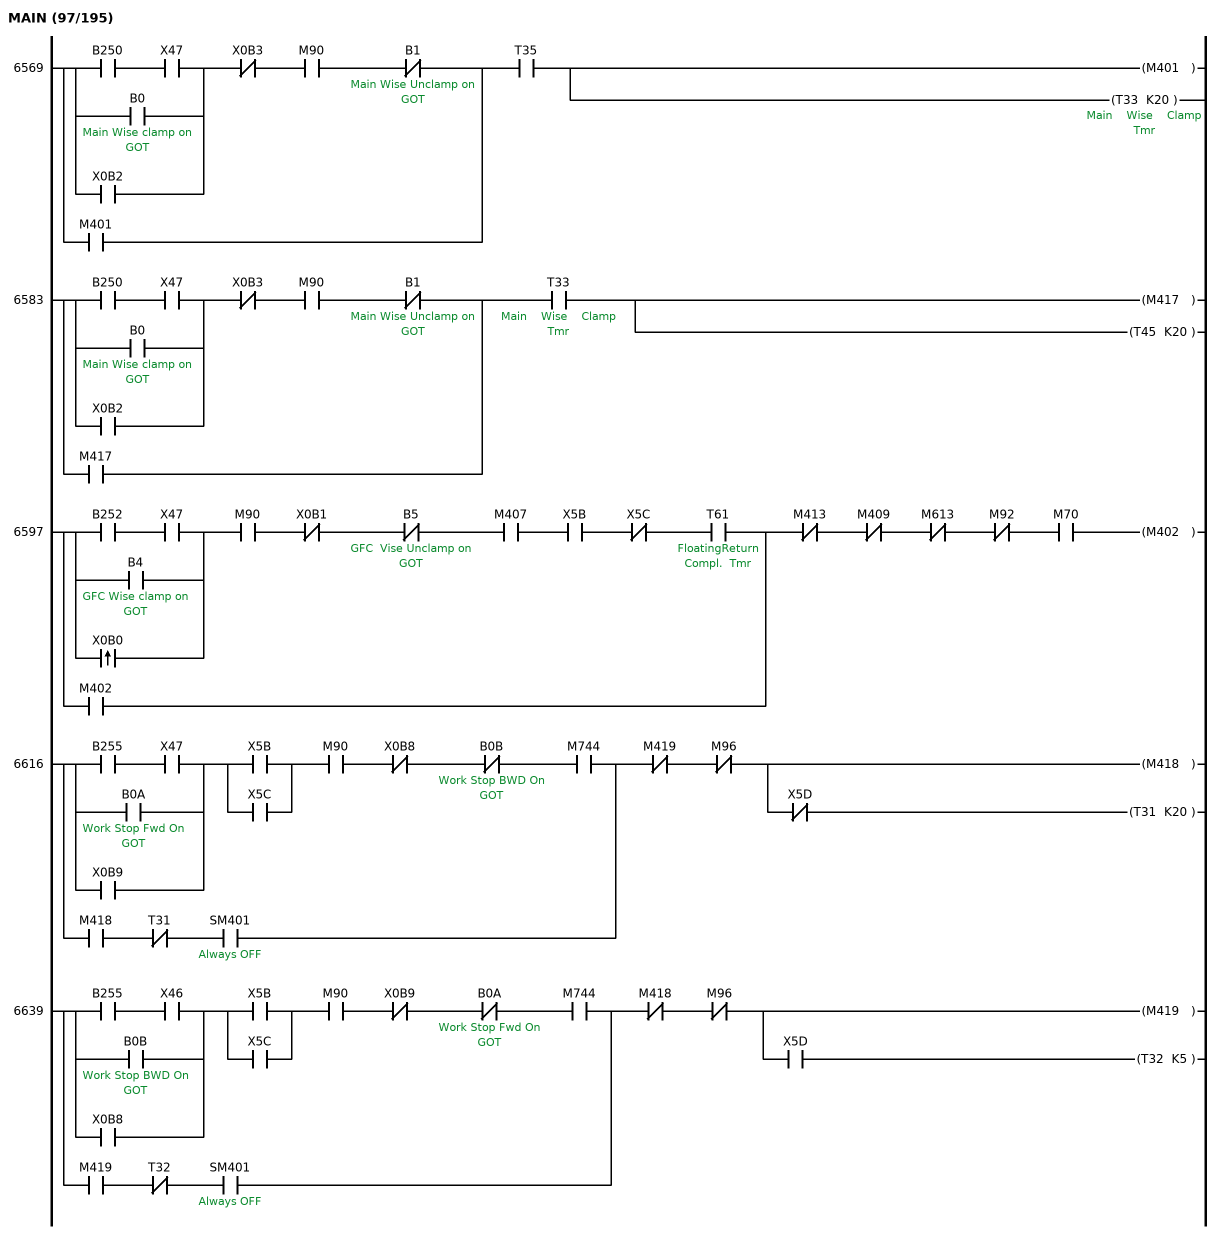
[picture p96: ladder of MAIN, rungs at steps 6569 to 6639]
6569  LD      B250
      AND     X47
      OR      B0  ; Main Wise clamp on GOT
      OR      X0B2
      ANI     X0B3
      AND     M90
      ANI     B1  ; Main Wise Unclamp on GOT
      OR      M401
      AND     T35
      OUT     M401
      OUT     T33 K20  ; Main    Wise    Clamp   Tmr
6583  LD      B250
      AND     X47
      OR      B0  ; Main Wise clamp on GOT
      OR      X0B2
      ANI     X0B3
      AND     M90
      ANI     B1  ; Main Wise Unclamp on GOT
      OR      M417
      AND     T33  ; Main    Wise    Clamp   Tmr
      OUT     M417
      OUT     T45 K20
6597  LD      B252
      AND     X47
      OR      B4  ; GFC Wise clamp on GOT
      ORP     X0B0
      AND     M90
      ANI     X0B1
      ANI     B5  ; GFC  Vise Unclamp on GOT
      AND     M407
      AND     X5B
      ANI     X5C
      AND     T61  ; FloatingReturn  Compl.  Tmr
      OR      M402
      ANI     M413
      ANI     M409
      ANI     M613
      ANI     M92
      AND     M70
      OUT     M402
6616  LD      B255
      AND     X47
      OR      B0A  ; Work Stop Fwd On GOT
      OR      X0B9
      LD      X5B
      OR      X5C
      ANB
      AND     M90
      ANI     X0B8
      ANI     B0B  ; Work Stop BWD On GOT
      AND     M744
      LD      M418
      ANI     T31
      AND     SM401  ; Always OFF
      ORB
      ANI     M419
      ANI     M96
      OUT     M418
      ANI     X5D
      OUT     T31 K20
6639  LD      B255
      AND     X46
      OR      B0B  ; Work Stop BWD On GOT
      OR      X0B8
      LD      X5B
      OR      X5C
      ANB
      AND     M90
      ANI     X0B9
      ANI     B0A  ; Work Stop Fwd On GOT
      AND     M744
      LD      M419
      ANI     T32
      AND     SM401  ; Always OFF
      ORB
      ANI     M418
      ANI     M96
      OUT     M419
      AND     X5D
      OUT     T32 K5
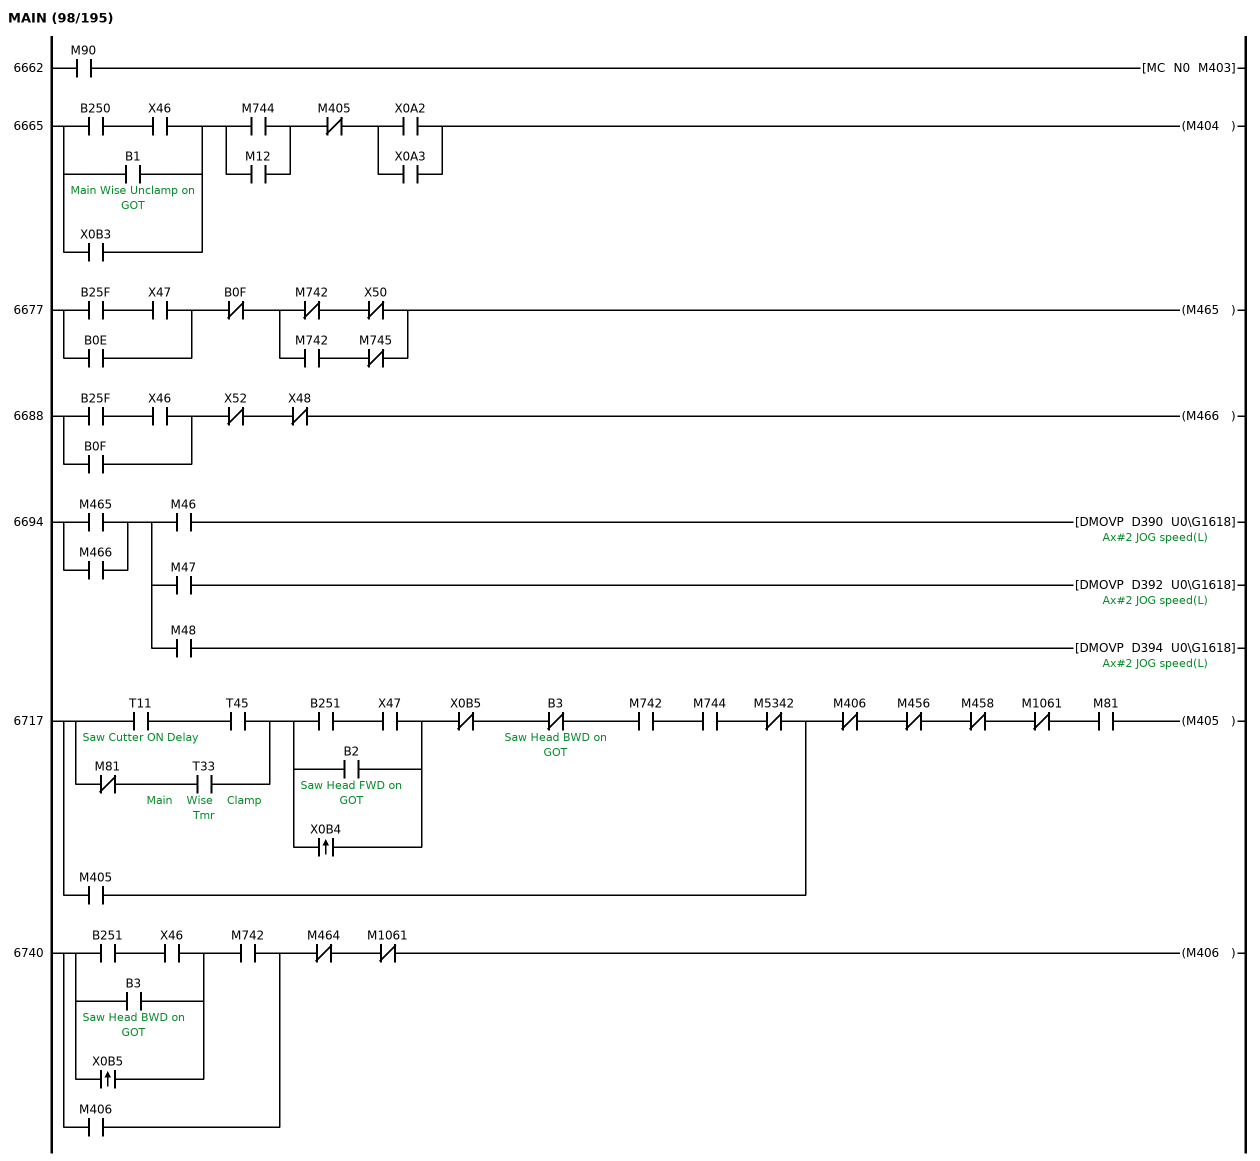
6662  LD      M90
      MC      N0 M403
6665  LD      B250
      AND     X46
      OR      B1  ; Main Wise Unclamp on GOT
      OR      X0B3
      LD      M744
      OR      M12
      ANB
      ANI     M405
      LD      X0A2
      OR      X0A3
      ANB
      OUT     M404
6677  LD      B25F
      AND     X47
      OR      B0E
      ANI     B0F
      LDI     M742
      ANI     X50
      LD      M742
      ANI     M745
      ORB
      ANB
      OUT     M465
6688  LD      B25F
      AND     X46
      OR      B0F
      ANI     X52
      ANI     X48
      OUT     M466
6694  LD      M465
      OR      M466
      MPS
      AND     M46
      DMOVP   D390 U0\G1618
      MRD
      AND     M47
      DMOVP   D392 U0\G1618
      MPP
      AND     M48
      DMOVP   D394 U0\G1618
6717  LD      T11  ; Saw Cutter ON Delay
      AND     T45
      LDI     M81
      AND     T33  ; Main    Wise    Clamp   Tmr
      ORB
      LD      B251
      AND     X47
      OR      B2  ; Saw Head FWD on GOT
      ORP     X0B4
      ANB
      ANI     X0B5
      ANI     B3  ; Saw Head BWD on GOT
      AND     M742
      AND     M744
      ANI     M5342
      OR      M405
      ANI     M406
      ANI     M456
      ANI     M458
      ANI     M1061
      AND     M81
      OUT     M405
6740  LD      B251
      AND     X46
      OR      B3  ; Saw Head BWD on GOT
      ORP     X0B5
      AND     M742
      OR      M406
      ANI     M464
      ANI     M1061
      OUT     M406
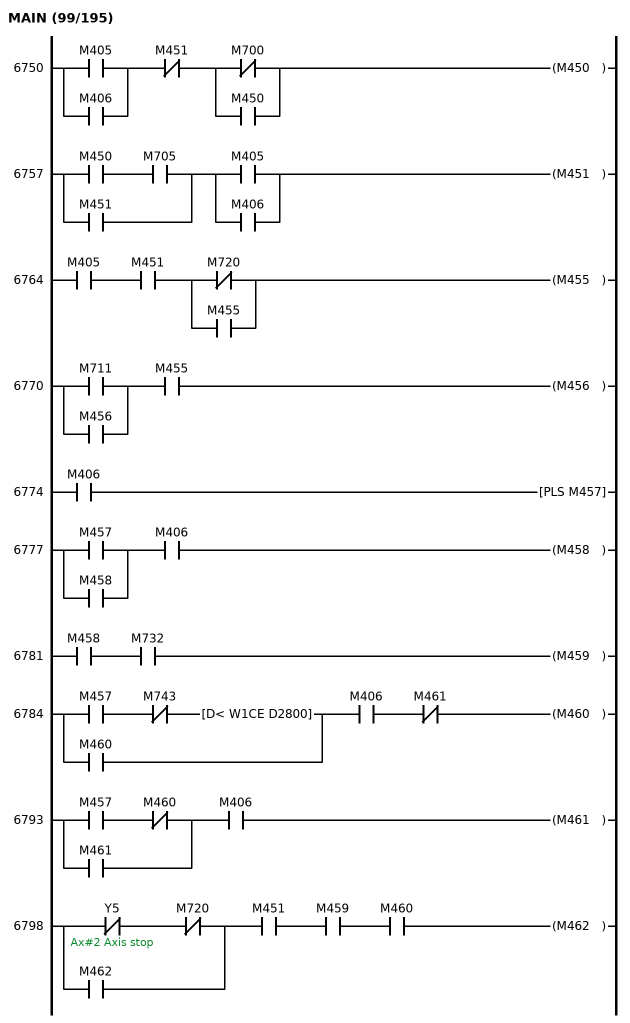
6750  LD      M405
      OR      M406
      ANI     M451
      LDI     M700
      OR      M450
      ANB
      OUT     M450
6757  LD      M450
      AND     M705
      OR      M451
      LD      M405
      OR      M406
      ANB
      OUT     M451
6764  LD      M405
      AND     M451
      LDI     M720
      OR      M455
      ANB
      OUT     M455
6770  LD      M711
      OR      M456
      AND     M455
      OUT     M456
6774  LD      M406
      PLS     M457
6777  LD      M457
      OR      M458
      AND     M406
      OUT     M458
6781  LD      M458
      AND     M732
      OUT     M459
6784  LD      M457
      ANI     M743
      ANDD<   W1CE D2800
      OR      M460
      AND     M406
      ANI     M461
      OUT     M460
6793  LD      M457
      ANI     M460
      OR      M461
      AND     M406
      OUT     M461
6798  LDI     Y5  ; Ax#2 Axis stop
      ANI     M720
      OR      M462
      AND     M451
      AND     M459
      AND     M460
      OUT     M462
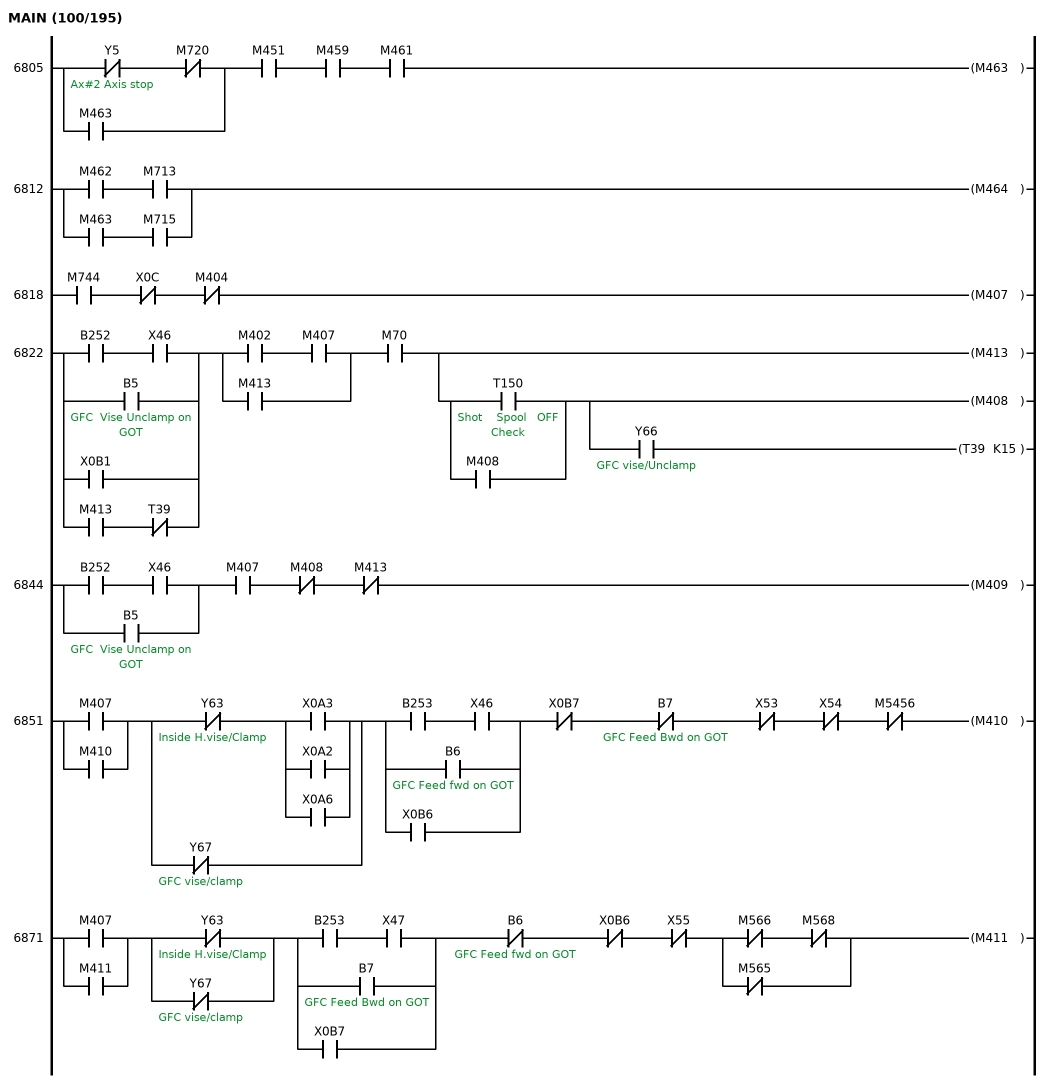
6805  LDI     Y5  ; Ax#2 Axis stop
      ANI     M720
      OR      M463
      AND     M451
      AND     M459
      AND     M461
      OUT     M463
6812  LD      M462
      AND     M713
      LD      M463
      AND     M715
      ORB
      OUT     M464
6818  LD      M744
      ANI     X0C
      ANI     M404
      OUT     M407
6822  LD      B252
      AND     X46
      OR      B5  ; GFC  Vise Unclamp on GOT
      OR      X0B1
      LD      M413
      ANI     T39
      ORB
      LD      M402
      AND     M407
      OR      M413
      ANB
      AND     M70
      OUT     M413
      LD      T150  ; Shot    Spool   OFF     Check
      OR      M408
      ANB
      OUT     M408
      AND     Y66  ; GFC vise/Unclamp
      OUT     T39 K15
6844  LD      B252
      AND     X46
      OR      B5  ; GFC  Vise Unclamp on GOT
      AND     M407
      ANI     M408
      ANI     M413
      OUT     M409
6851  LD      M407
      OR      M410
      LDI     Y63  ; Inside H.vise/Clamp
      LD      X0A3
      OR      X0A2
      OR      X0A6
      ANB
      ORI     Y67  ; GFC vise/clamp
      ANB
      LD      B253
      AND     X46
      OR      B6  ; GFC Feed fwd on GOT
      OR      X0B6
      ANB
      ANI     X0B7
      ANI     B7  ; GFC Feed Bwd on GOT
      ANI     X53
      ANI     X54
      ANI     M5456
      OUT     M410
6871  LD      M407
      OR      M411
      LDI     Y63  ; Inside H.vise/Clamp
      ORI     Y67  ; GFC vise/clamp
      ANB
      LD      B253
      AND     X47
      OR      B7  ; GFC Feed Bwd on GOT
      OR      X0B7
      ANB
      ANI     B6  ; GFC Feed fwd on GOT
      ANI     X0B6
      ANI     X55
      LDI     M566
      ANI     M568
      ORI     M565
      ANB
      OUT     M411
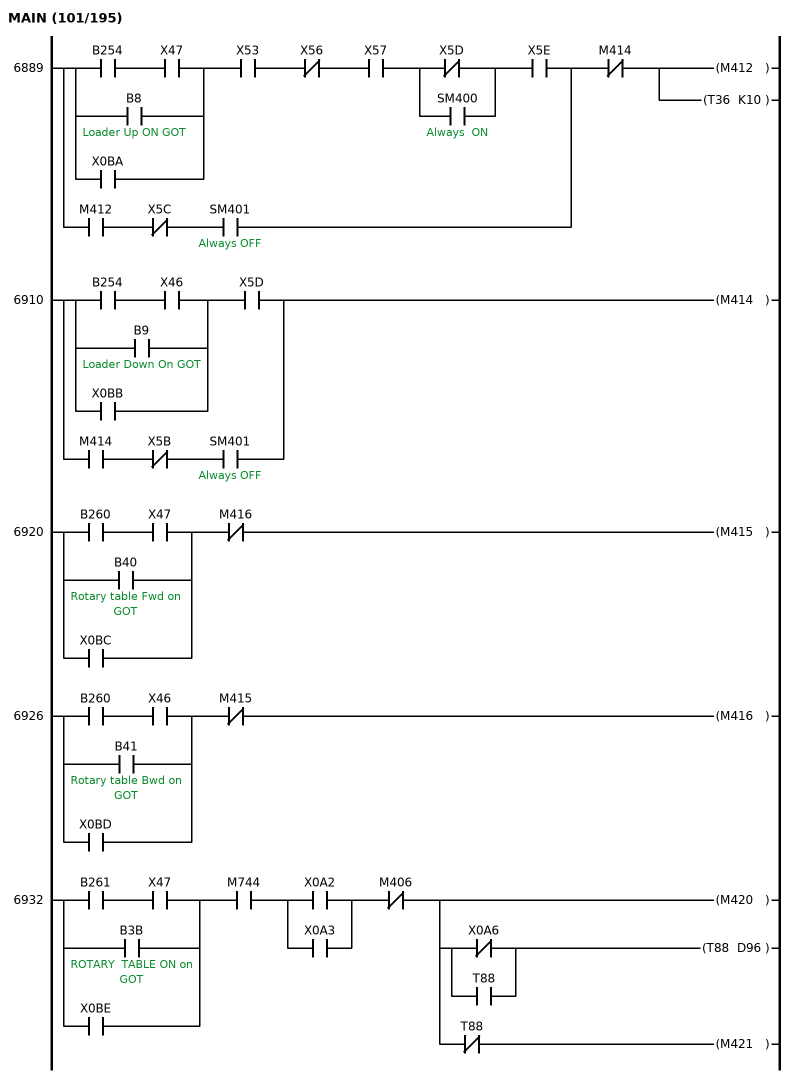
6889  LD      B254
      AND     X47
      OR      B8  ; Loader Up ON GOT
      OR      X0BA
      AND     X53
      ANI     X56
      AND     X57
      LDI     X5D
      OR      SM400  ; Always  ON
      ANB
      AND     X5E
      LD      M412
      ANI     X5C
      AND     SM401  ; Always OFF
      ORB
      ANI     M414
      OUT     M412
      OUT     T36 K10
6910  LD      B254
      AND     X46
      OR      B9  ; Loader Down On GOT
      OR      X0BB
      AND     X5D
      LD      M414
      ANI     X5B
      AND     SM401  ; Always OFF
      ORB
      OUT     M414
6920  LD      B260
      AND     X47
      OR      B40  ; Rotary table Fwd on GOT
      OR      X0BC
      ANI     M416
      OUT     M415
6926  LD      B260
      AND     X46
      OR      B41  ; Rotary table Bwd on GOT
      OR      X0BD
      ANI     M415
      OUT     M416
6932  LD      B261
      AND     X47
      OR      B3B  ; ROTARY  TABLE ON on GOT
      OR      X0BE
      AND     M744
      LD      X0A2
      OR      X0A3
      ANB
      ANI     M406
      OUT     M420
      MPS
      LDI     X0A6
      OR      T88
      ANB
      OUT     T88 D96
      MPP
      ANI     T88
      OUT     M421
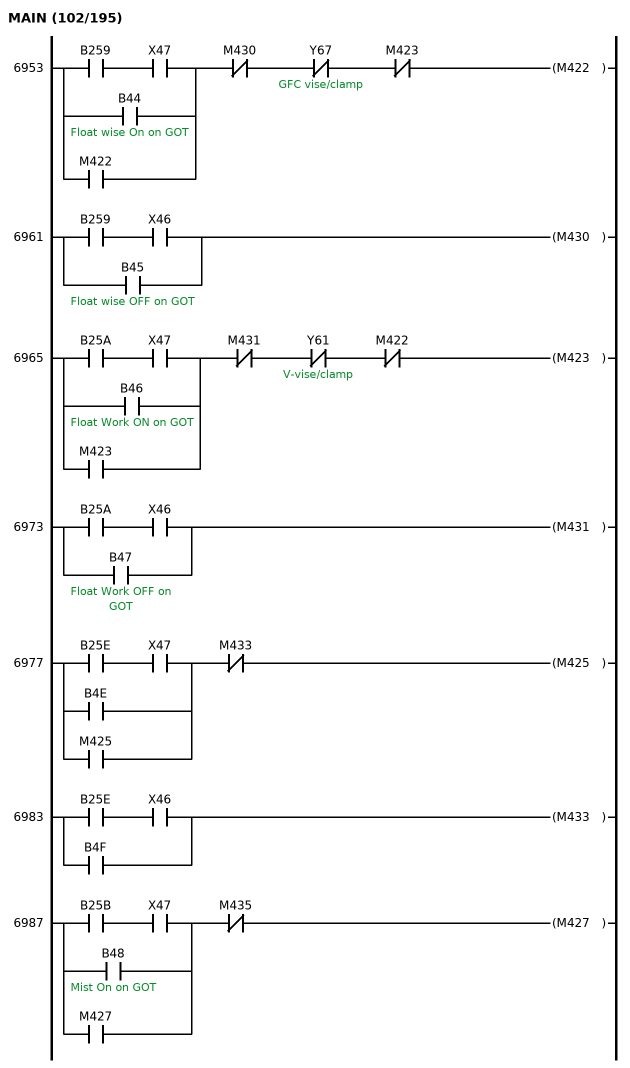
6953  LD      B259
      AND     X47
      OR      B44  ; Float wise On on GOT
      OR      M422
      ANI     M430
      ANI     Y67  ; GFC vise/clamp
      ANI     M423
      OUT     M422
6961  LD      B259
      AND     X46
      OR      B45  ; Float wise OFF on GOT
      OUT     M430
6965  LD      B25A
      AND     X47
      OR      B46  ; Float Work ON on GOT
      OR      M423
      ANI     M431
      ANI     Y61  ; V-vise/clamp
      ANI     M422
      OUT     M423
6973  LD      B25A
      AND     X46
      OR      B47  ; Float Work OFF on GOT
      OUT     M431
6977  LD      B25E
      AND     X47
      OR      B4E
      OR      M425
      ANI     M433
      OUT     M425
6983  LD      B25E
      AND     X46
      OR      B4F
      OUT     M433
6987  LD      B25B
      AND     X47
      OR      B48  ; Mist On on GOT
      OR      M427
      ANI     M435
      OUT     M427
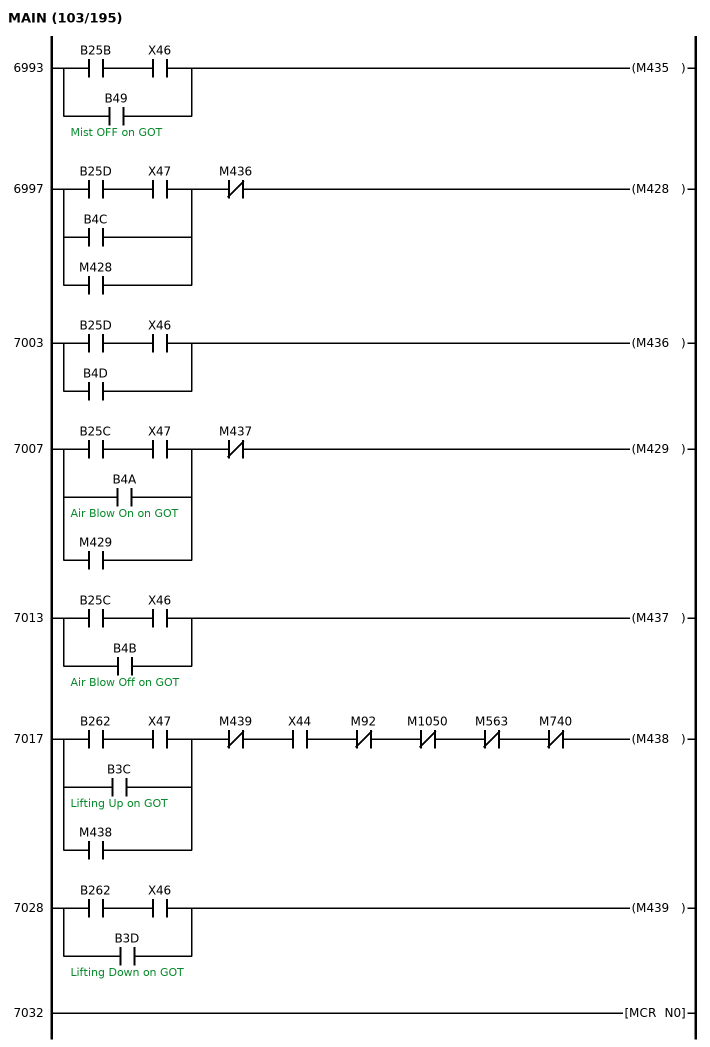
6993  LD      B25B
      AND     X46
      OR      B49  ; Mist OFF on GOT
      OUT     M435
6997  LD      B25D
      AND     X47
      OR      B4C
      OR      M428
      ANI     M436
      OUT     M428
7003  LD      B25D
      AND     X46
      OR      B4D
      OUT     M436
7007  LD      B25C
      AND     X47
      OR      B4A  ; Air Blow On on GOT
      OR      M429
      ANI     M437
      OUT     M429
7013  LD      B25C
      AND     X46
      OR      B4B  ; Air Blow Off on GOT
      OUT     M437
7017  LD      B262
      AND     X47
      OR      B3C  ; Lifting Up on GOT
      OR      M438
      ANI     M439
      AND     X44
      ANI     M92
      ANI     M1050
      ANI     M563
      ANI     M740
      OUT     M438
7028  LD      B262
      AND     X46
      OR      B3D  ; Lifting Down on GOT
      OUT     M439
7032  MCR     N0
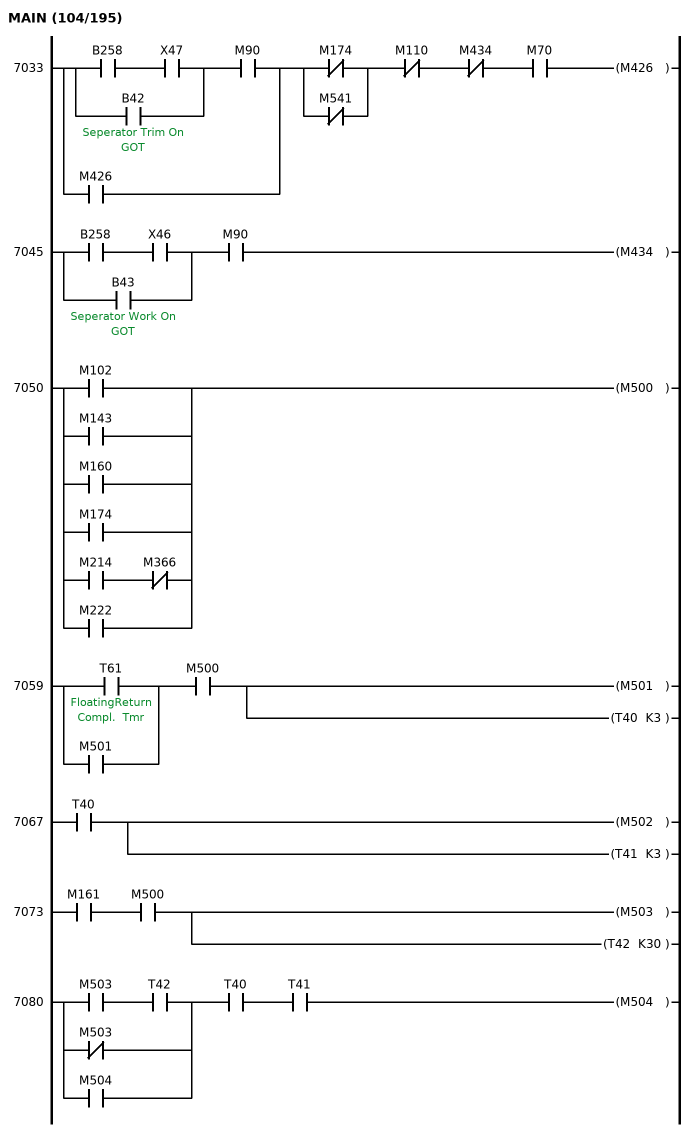
7033  LD      B258
      AND     X47
      OR      B42  ; Seperator Trim On GOT
      AND     M90
      OR      M426
      LDI     M174
      ORI     M541
      ANB
      ANI     M110
      ANI     M434
      AND     M70
      OUT     M426
7045  LD      B258
      AND     X46
      OR      B43  ; Seperator Work On GOT
      AND     M90
      OUT     M434
7050  LD      M102
      OR      M143
      OR      M160
      OR      M174
      LD      M214
      ANI     M366
      ORB
      OR      M222
      OUT     M500
7059  LD      T61  ; FloatingReturn  Compl.  Tmr
      OR      M501
      AND     M500
      OUT     M501
      OUT     T40 K3
7067  LD      T40
      OUT     M502
      OUT     T41 K3
7073  LD      M161
      AND     M500
      OUT     M503
      OUT     T42 K30
7080  LD      M503
      AND     T42
      ORI     M503
      OR      M504
      AND     T40
      AND     T41
      OUT     M504
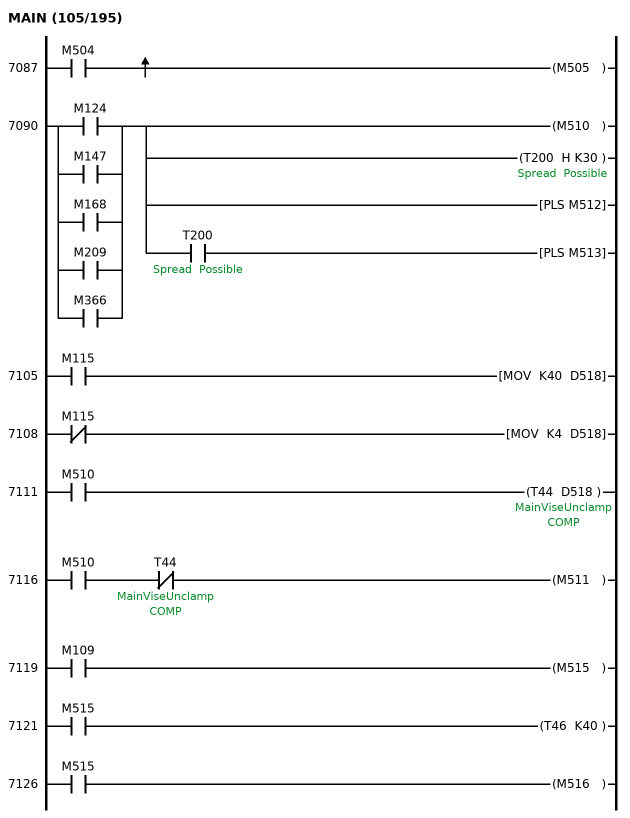
7087  LD      M504
      MEP
      OUT     M505
7090  LD      M124
      OR      M147
      OR      M168
      OR      M209
      OR      M366
      OUT     M510
      OUTH    T200 K30  ; Spread  Possible
      PLS     M512
      AND     T200  ; Spread  Possible
      PLS     M513
7105  LD      M115
      MOV     K40 D518
7108  LDI     M115
      MOV     K4 D518
7111  LD      M510
      OUT     T44 D518  ; MainViseUnclamp COMP
7116  LD      M510
      ANI     T44  ; MainViseUnclamp COMP
      OUT     M511
7119  LD      M109
      OUT     M515
7121  LD      M515
      OUT     T46 K40
7126  LD      M515
      OUT     M516
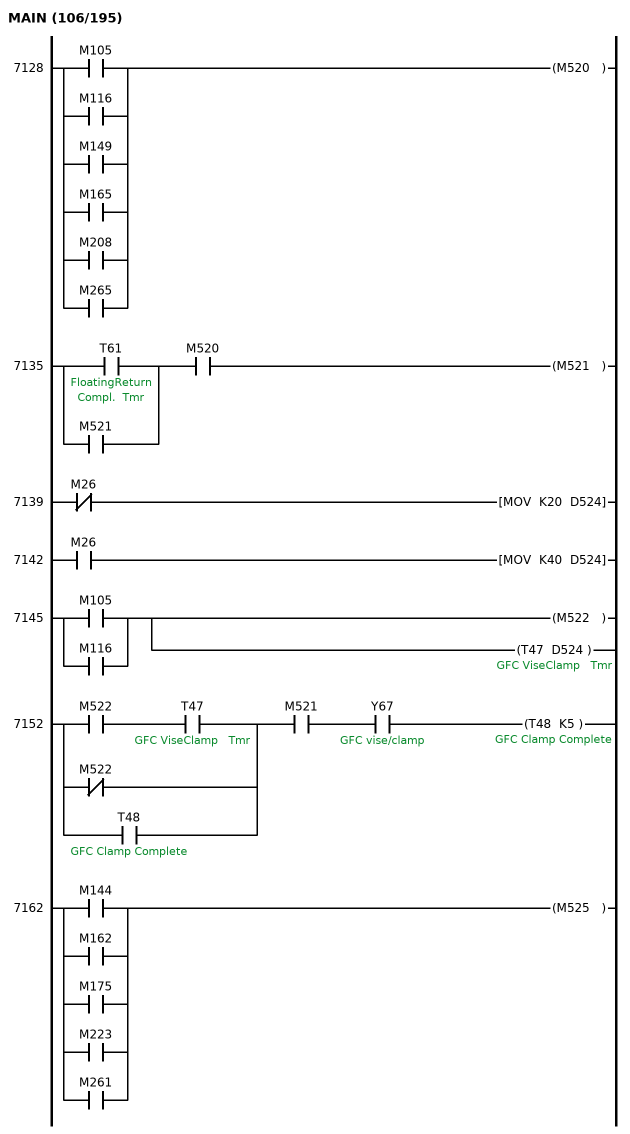
7128  LD      M105
      OR      M116
      OR      M149
      OR      M165
      OR      M208
      OR      M265
      OUT     M520
7135  LD      T61  ; FloatingReturn  Compl.  Tmr
      OR      M521
      AND     M520
      OUT     M521
7139  LDI     M26
      MOV     K20 D524
7142  LD      M26
      MOV     K40 D524
7145  LD      M105
      OR      M116
      OUT     M522
      OUT     T47 D524  ; GFC ViseClamp   Tmr
7152  LD      M522
      AND     T47  ; GFC ViseClamp   Tmr
      ORI     M522
      OR      T48  ; GFC Clamp Complete
      AND     M521
      AND     Y67  ; GFC vise/clamp
      OUT     T48 K5  ; GFC Clamp Complete
7162  LD      M144
      OR      M162
      OR      M175
      OR      M223
      OR      M261
      OUT     M525
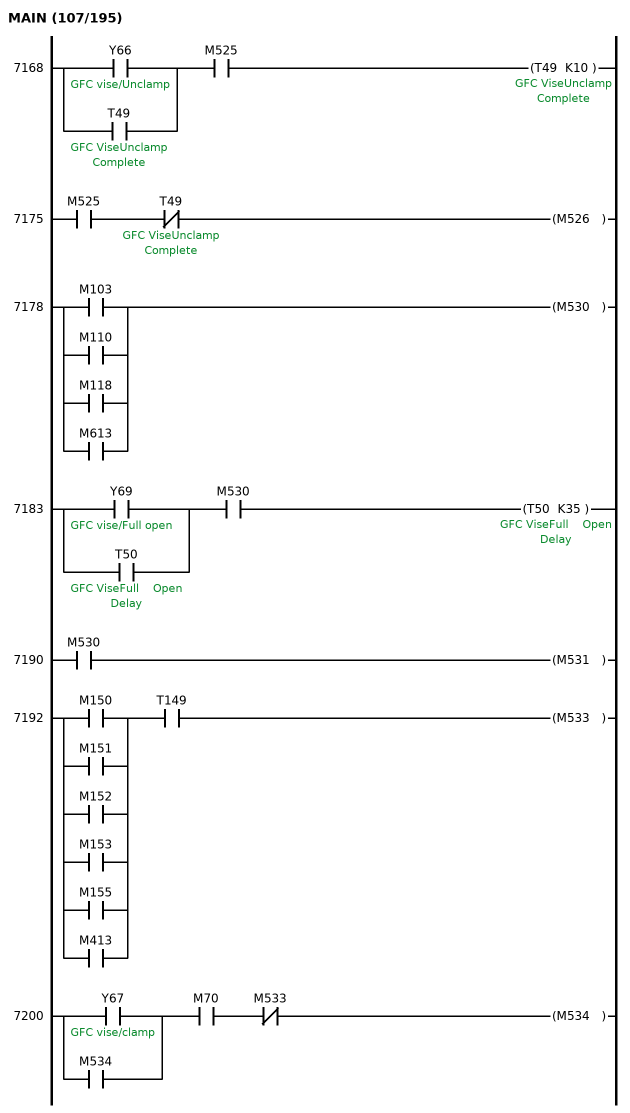
7168  LD      Y66  ; GFC vise/Unclamp
      OR      T49  ; GFC ViseUnclamp Complete
      AND     M525
      OUT     T49 K10  ; GFC ViseUnclamp Complete
7175  LD      M525
      ANI     T49  ; GFC ViseUnclamp Complete
      OUT     M526
7178  LD      M103
      OR      M110
      OR      M118
      OR      M613
      OUT     M530
7183  LD      Y69  ; GFC vise/Full open
      OR      T50  ; GFC ViseFull    Open    Delay
      AND     M530
      OUT     T50 K35  ; GFC ViseFull    Open    Delay
7190  LD      M530
      OUT     M531
7192  LD      M150
      OR      M151
      OR      M152
      OR      M153
      OR      M155
      OR      M413
      AND     T149
      OUT     M533
7200  LD      Y67  ; GFC vise/clamp
      OR      M534
      AND     M70
      ANI     M533
      OUT     M534
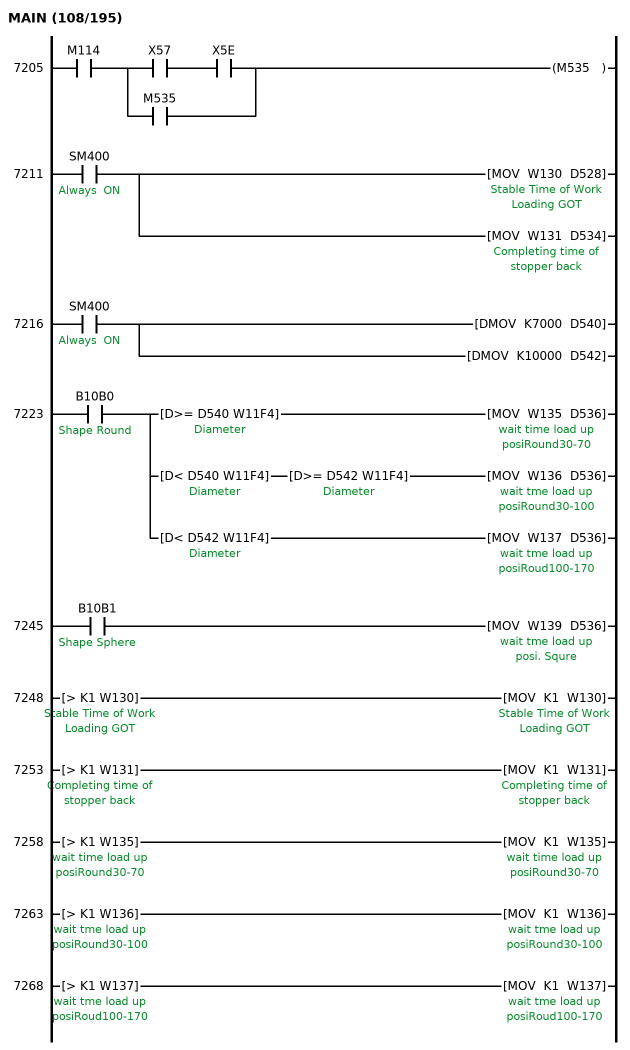
7205  LD      M114
      LD      X57
      AND     X5E
      OR      M535
      ANB
      OUT     M535
7211  LD      SM400  ; Always  ON
      MOV     W130 D528
      MOV     W131 D534  ; Completing time of stopper back
7216  LD      SM400  ; Always  ON
      DMOV    K7000 D540
      DMOV    K10000 D542
7223  LD      B10B0  ; Shape Round
      MPS
      ANDD>=  D540 W11F4  ; Diameter
      MOV     W135 D536  ; wait time load up posiRound30-70
      MRD
      ANDD<   D540 W11F4  ; Diameter
      ANDD>=  D542 W11F4  ; Diameter
      MOV     W136 D536  ; wait tme load up posiRound30-100
      MPP
      ANDD<   D542 W11F4  ; Diameter
      MOV     W137 D536  ; wait tme load up posiRoud100-170
7245  LD      B10B1  ; Shape Sphere
      MOV     W139 D536  ; wait tme load up posi. Squre
7248  LD>     K1 W130  ; Stable Time of Work Loading GOT
      MOV     K1 W130
7253  LD>     K1 W131  ; Completing time of stopper back
      MOV     K1 W131
7258  LD>     K1 W135  ; wait time load up posiRound30-70
      MOV     K1 W135
7263  LD>     K1 W136  ; wait tme load up posiRound30-100
      MOV     K1 W136
7268  LD>     K1 W137  ; wait tme load up posiRoud100-170
      MOV     K1 W137
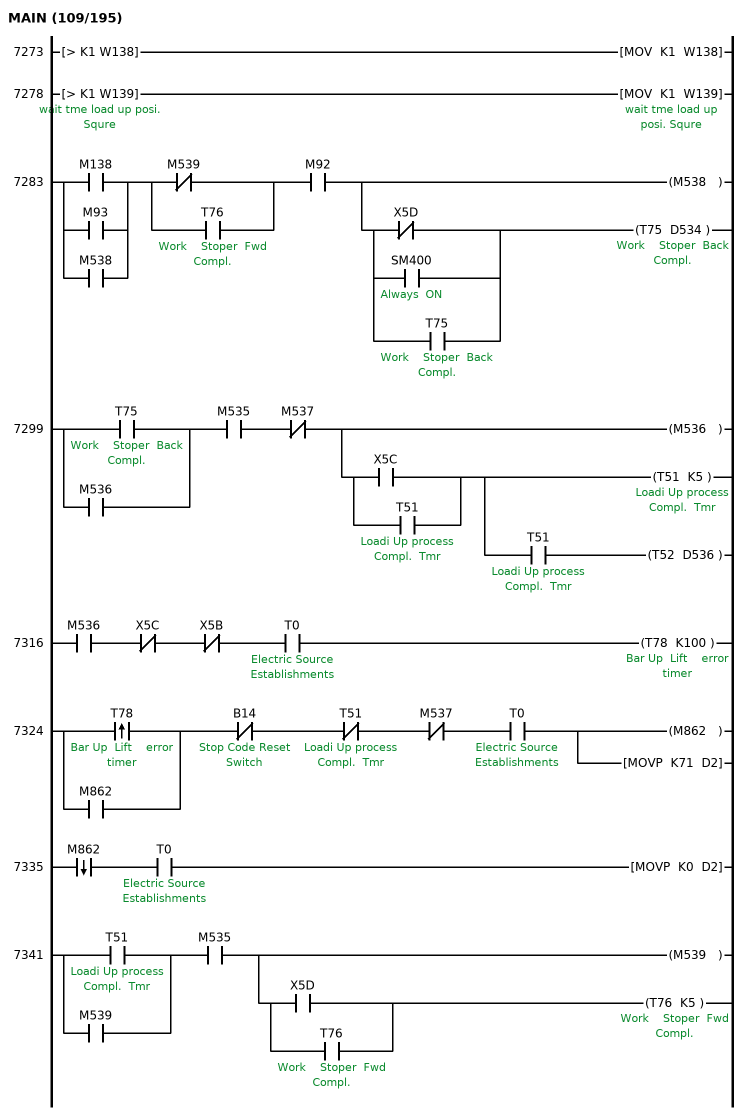
7273  LD>     K1 W138
      MOV     K1 W138
7278  LD>     K1 W139  ; wait tme load up posi. Squre
      MOV     K1 W139
7283  LD      M138
      OR      M93
      OR      M538
      LDI     M539
      OR      T76  ; Work    Stoper  Fwd     Compl.
      ANB
      AND     M92
      OUT     M538
      LDI     X5D
      OR      SM400  ; Always  ON
      OR      T75  ; Work    Stoper  Back    Compl.
      ANB
      OUT     T75 D534  ; Work    Stoper  Back    Compl.
7299  LD      T75  ; Work    Stoper  Back    Compl.
      OR      M536
      AND     M535
      ANI     M537
      OUT     M536
      LD      X5C
      OR      T51  ; Loadi Up process Compl.  Tmr
      ANB
      OUT     T51 K5  ; Loadi Up process Compl.  Tmr
      AND     T51  ; Loadi Up process Compl.  Tmr
      OUT     T52 D536
7316  LD      M536
      ANI     X5C
      ANI     X5B
      AND     T0  ; Electric Source Establishments
      OUT     T78 K100  ; Bar Up  Lift    error   timer
7324  LDP     T78  ; Bar Up  Lift    error   timer
      OR      M862
      ANI     B14  ; Stop Code Reset Switch
      ANI     T51  ; Loadi Up process Compl.  Tmr
      ANI     M537
      AND     T0  ; Electric Source Establishments
      OUT     M862
      MOVP    K71 D2
7335  LDF     M862
      AND     T0  ; Electric Source Establishments
      MOVP    K0 D2
7341  LD      T51  ; Loadi Up process Compl.  Tmr
      OR      M539
      AND     M535
      OUT     M539
      LD      X5D
      OR      T76  ; Work    Stoper  Fwd     Compl.
      ANB
      OUT     T76 K5  ; Work    Stoper  Fwd     Compl.
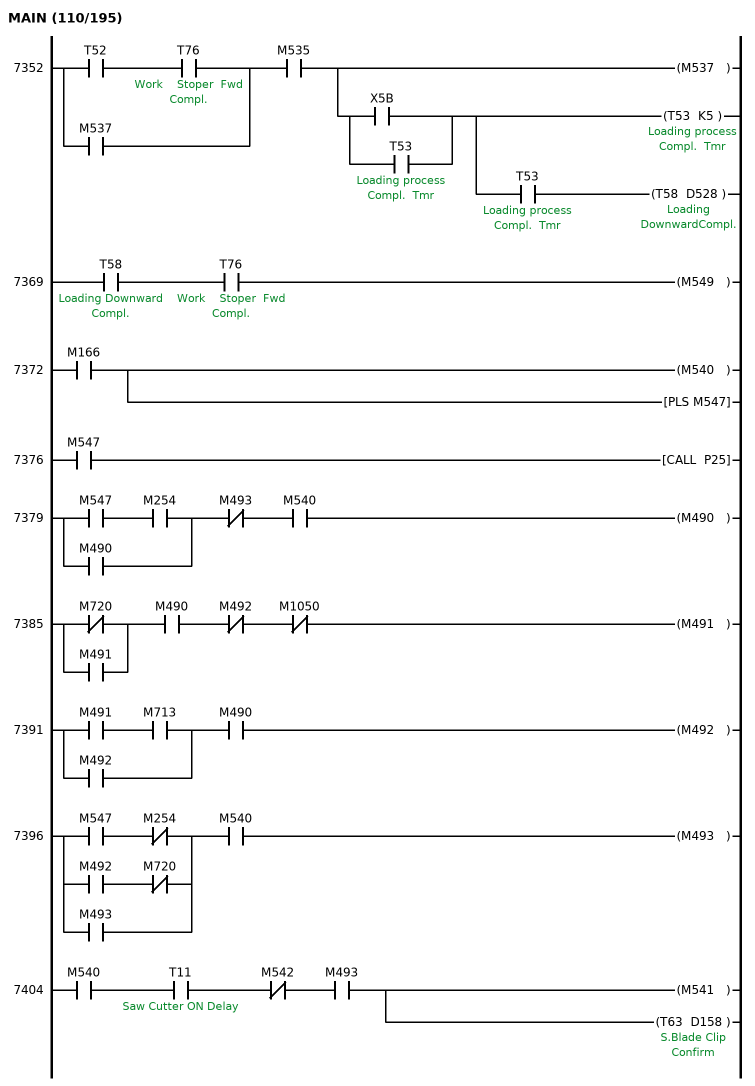
7352  LD      T52
      AND     T76  ; Work    Stoper  Fwd     Compl.
      OR      M537
      AND     M535
      OUT     M537
      LD      X5B
      OR      T53  ; Loading process Compl.  Tmr
      ANB
      OUT     T53 K5  ; Loading process Compl.  Tmr
      AND     T53  ; Loading process Compl.  Tmr
      OUT     T58 D528  ; Loading DownwardCompl.
7369  LD      T58  ; Loading DownwardCompl.
      AND     T76  ; Work    Stoper  Fwd     Compl.
      OUT     M549
7372  LD      M166
      OUT     M540
      PLS     M547
7376  LD      M547
      CALL    P25
7379  LD      M547
      AND     M254
      OR      M490
      ANI     M493
      AND     M540
      OUT     M490
7385  LDI     M720
      OR      M491
      AND     M490
      ANI     M492
      ANI     M1050
      OUT     M491
7391  LD      M491
      AND     M713
      OR      M492
      AND     M490
      OUT     M492
7396  LD      M547
      ANI     M254
      LD      M492
      ANI     M720
      ORB
      OR      M493
      AND     M540
      OUT     M493
7404  LD      M540
      AND     T11  ; Saw Cutter ON Delay
      ANI     M542
      AND     M493
      OUT     M541
      OUT     T63 D158  ; S.Blade Clip    Confirm
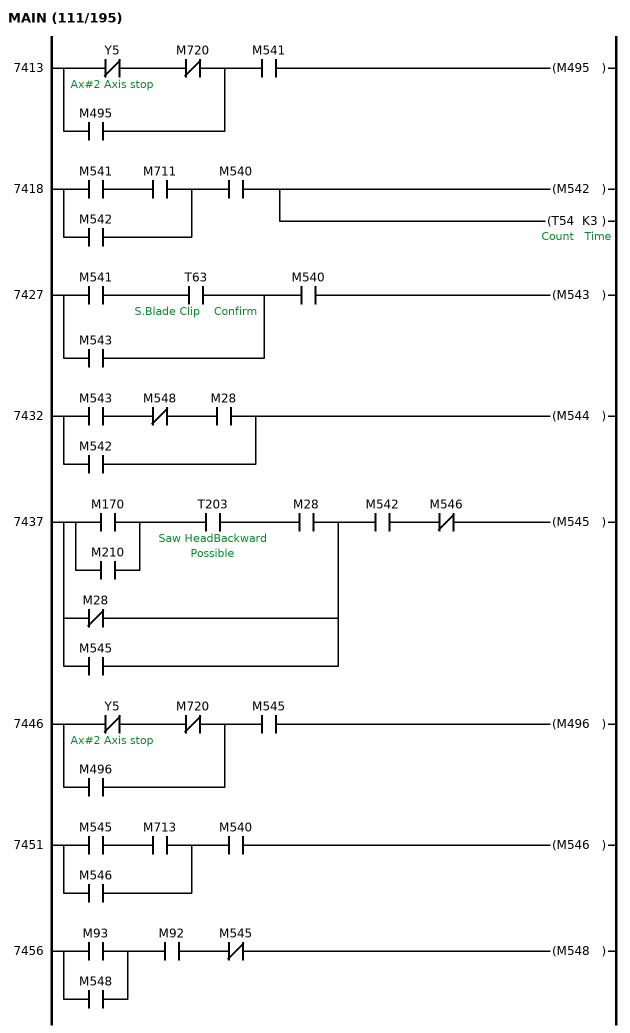
7413  LDI     Y5  ; Ax#2 Axis stop
      ANI     M720
      OR      M495
      AND     M541
      OUT     M495
7418  LD      M541
      AND     M711
      OR      M542
      AND     M540
      OUT     M542
      OUT     T54 K3  ; Count   Time
7427  LD      M541
      AND     T63  ; S.Blade Clip    Confirm
      OR      M543
      AND     M540
      OUT     M543
7432  LD      M543
      ANI     M548
      AND     M28
      OR      M542
      OUT     M544
7437  LD      M170
      OR      M210
      AND     T203  ; Saw HeadBackwardPossible
      AND     M28
      ORI     M28
      OR      M545
      AND     M542
      ANI     M546
      OUT     M545
7446  LDI     Y5  ; Ax#2 Axis stop
      ANI     M720
      OR      M496
      AND     M545
      OUT     M496
7451  LD      M545
      AND     M713
      OR      M546
      AND     M540
      OUT     M546
7456  LD      M93
      OR      M548
      AND     M92
      ANI     M545
      OUT     M548
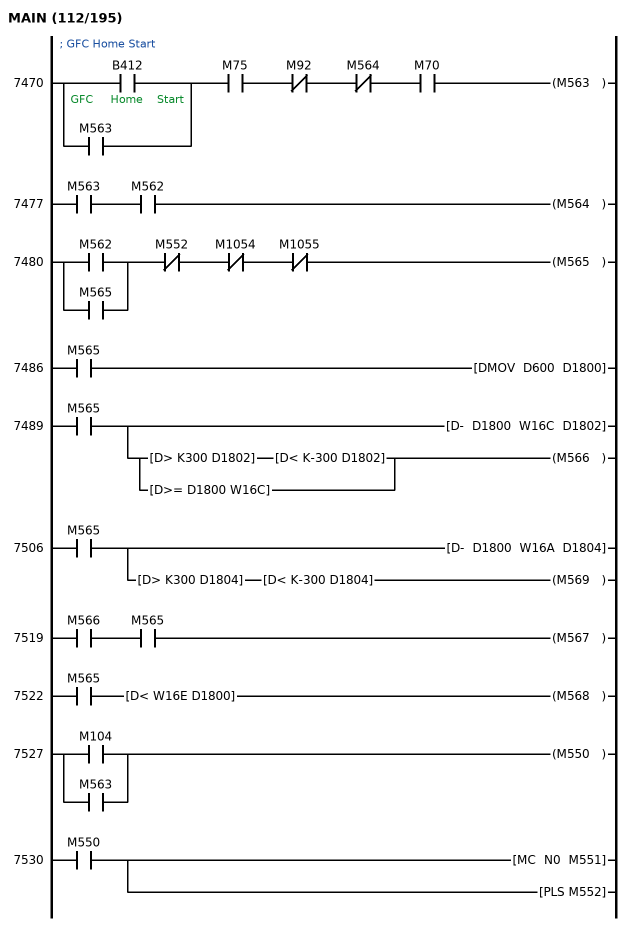
; GFC Home Start
7470  LD      B412  ; GFC     Home    Start
      OR      M563
      AND     M75
      ANI     M92
      ANI     M564
      AND     M70
      OUT     M563
7477  LD      M563
      AND     M562
      OUT     M564
7480  LD      M562
      OR      M565
      ANI     M552
      ANI     M1054
      ANI     M1055
      OUT     M565
7486  LD      M565
      DMOV    D600 D1800
7489  LD      M565
      D-      D1800 W16C D1802
      LDD>    K300 D1802
      ANDD<   K-300 D1802
      ORD>=   D1800 W16C
      ANB
      OUT     M566
7506  LD      M565
      D-      D1800 W16A D1804
      ANDD>   K300 D1804
      ANDD<   K-300 D1804
      OUT     M569
7519  LD      M566
      AND     M565
      OUT     M567
7522  LD      M565
      ANDD<   W16E D1800
      OUT     M568
7527  LD      M104
      OR      M563
      OUT     M550
7530  LD      M550
      MC      N0 M551
      PLS     M552
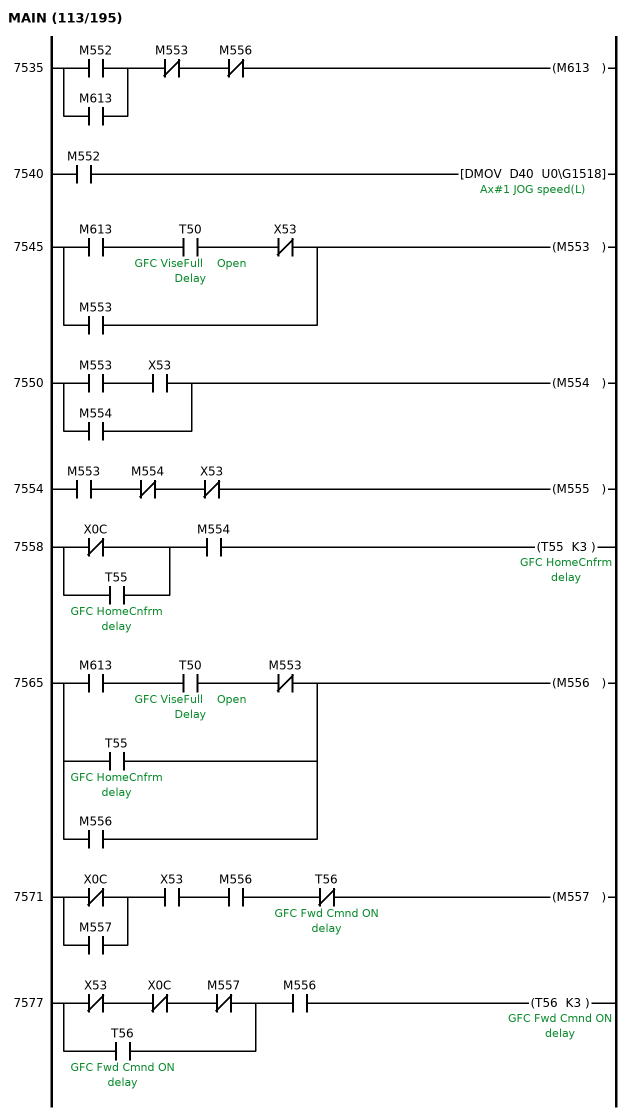
7535  LD      M552
      OR      M613
      ANI     M553
      ANI     M556
      OUT     M613
7540  LD      M552
      DMOV    D40 U0\G1518
7545  LD      M613
      AND     T50  ; GFC ViseFull    Open    Delay
      ANI     X53
      OR      M553
      OUT     M553
7550  LD      M553
      AND     X53
      OR      M554
      OUT     M554
7554  LD      M553
      ANI     M554
      ANI     X53
      OUT     M555
7558  LDI     X0C
      OR      T55  ; GFC HomeCnfrm   delay
      AND     M554
      OUT     T55 K3  ; GFC HomeCnfrm   delay
7565  LD      M613
      AND     T50  ; GFC ViseFull    Open    Delay
      ANI     M553
      OR      T55  ; GFC HomeCnfrm   delay
      OR      M556
      OUT     M556
7571  LDI     X0C
      OR      M557
      AND     X53
      AND     M556
      ANI     T56  ; GFC Fwd Cmnd ON delay
      OUT     M557
7577  LDI     X53
      ANI     X0C
      ANI     M557
      OR      T56  ; GFC Fwd Cmnd ON delay
      AND     M556
      OUT     T56 K3  ; GFC Fwd Cmnd ON delay
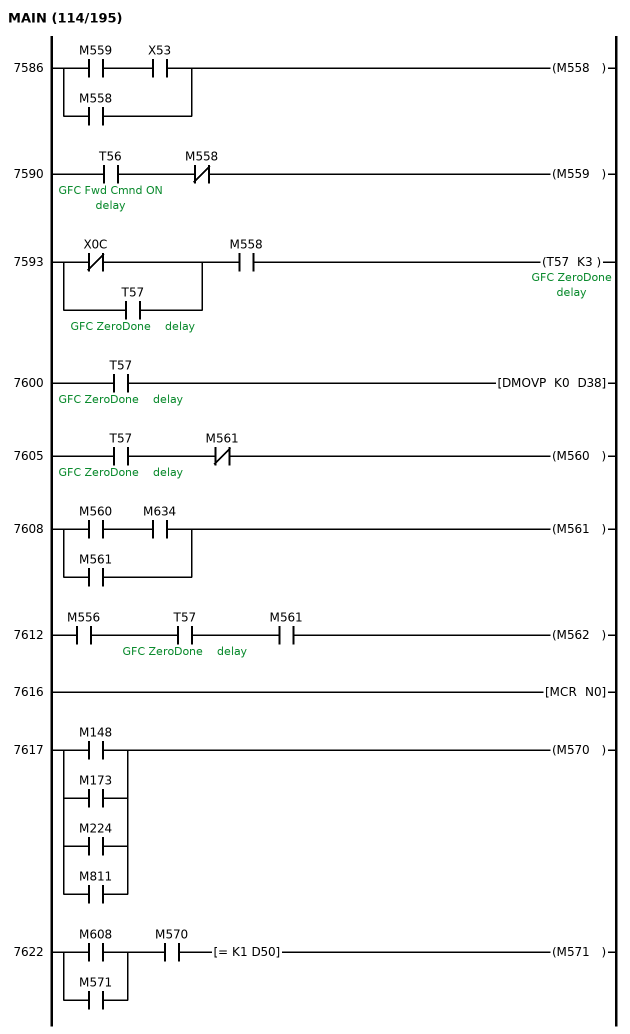
7586  LD      M559
      AND     X53
      OR      M558
      OUT     M558
7590  LD      T56  ; GFC Fwd Cmnd ON delay
      ANI     M558
      OUT     M559
7593  LDI     X0C
      OR      T57  ; GFC ZeroDone    delay
      AND     M558
      OUT     T57 K3  ; GFC ZeroDone    delay
7600  LD      T57  ; GFC ZeroDone    delay
      DMOVP   K0 D38
7605  LD      T57  ; GFC ZeroDone    delay
      ANI     M561
      OUT     M560
7608  LD      M560
      AND     M634
      OR      M561
      OUT     M561
7612  LD      M556
      AND     T57  ; GFC ZeroDone    delay
      AND     M561
      OUT     M562
7616  MCR     N0
7617  LD      M148
      OR      M173
      OR      M224
      OR      M811
      OUT     M570
7622  LD      M608
      OR      M571
      AND     M570
      AND=    K1 D50
      OUT     M571
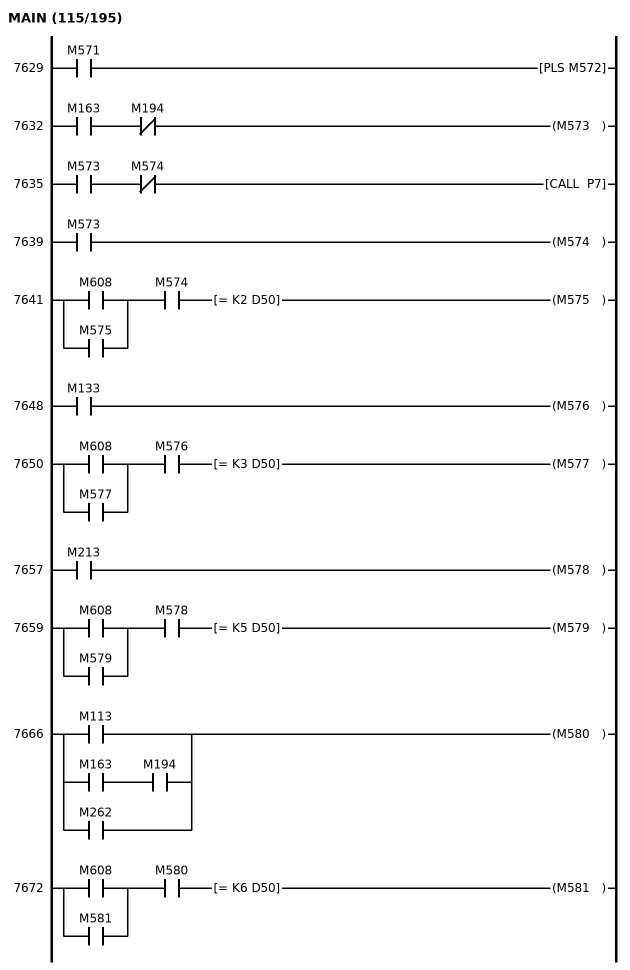
7629  LD      M571
      PLS     M572
7632  LD      M163
      ANI     M194
      OUT     M573
7635  LD      M573
      ANI     M574
      CALL    P7
7639  LD      M573
      OUT     M574
7641  LD      M608
      OR      M575
      AND     M574
      AND=    K2 D50
      OUT     M575
7648  LD      M133
      OUT     M576
7650  LD      M608
      OR      M577
      AND     M576
      AND=    K3 D50
      OUT     M577
7657  LD      M213
      OUT     M578
7659  LD      M608
      OR      M579
      AND     M578
      AND=    K5 D50
      OUT     M579
7666  LD      M113
      LD      M163
      AND     M194
      ORB
      OR      M262
      OUT     M580
7672  LD      M608
      OR      M581
      AND     M580
      AND=    K6 D50
      OUT     M581
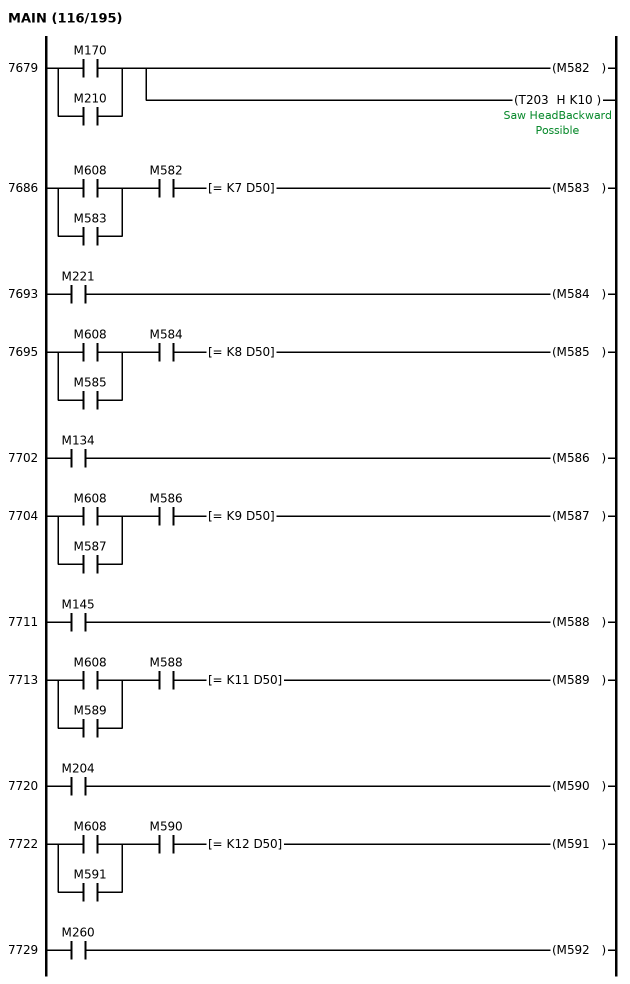
7679  LD      M170
      OR      M210
      OUT     M582
      OUTH    T203 K10  ; Saw HeadBackwardPossible
7686  LD      M608
      OR      M583
      AND     M582
      AND=    K7 D50
      OUT     M583
7693  LD      M221
      OUT     M584
7695  LD      M608
      OR      M585
      AND     M584
      AND=    K8 D50
      OUT     M585
7702  LD      M134
      OUT     M586
7704  LD      M608
      OR      M587
      AND     M586
      AND=    K9 D50
      OUT     M587
7711  LD      M145
      OUT     M588
7713  LD      M608
      OR      M589
      AND     M588
      AND=    K11 D50
      OUT     M589
7720  LD      M204
      OUT     M590
7722  LD      M608
      OR      M591
      AND     M590
      AND=    K12 D50
      OUT     M591
7729  LD      M260
      OUT     M592
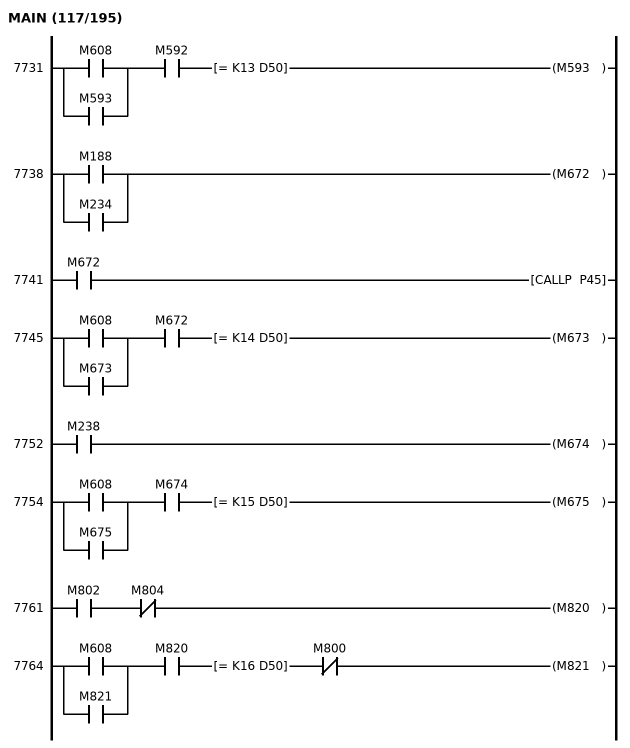
7731  LD      M608
      OR      M593
      AND     M592
      AND=    K13 D50
      OUT     M593
7738  LD      M188
      OR      M234
      OUT     M672
7741  LD      M672
      CALLP   P45
7745  LD      M608
      OR      M673
      AND     M672
      AND=    K14 D50
      OUT     M673
7752  LD      M238
      OUT     M674
7754  LD      M608
      OR      M675
      AND     M674
      AND=    K15 D50
      OUT     M675
7761  LD      M802
      ANI     M804
      OUT     M820
7764  LD      M608
      OR      M821
      AND     M820
      AND=    K16 D50
      ANI     M800
      OUT     M821
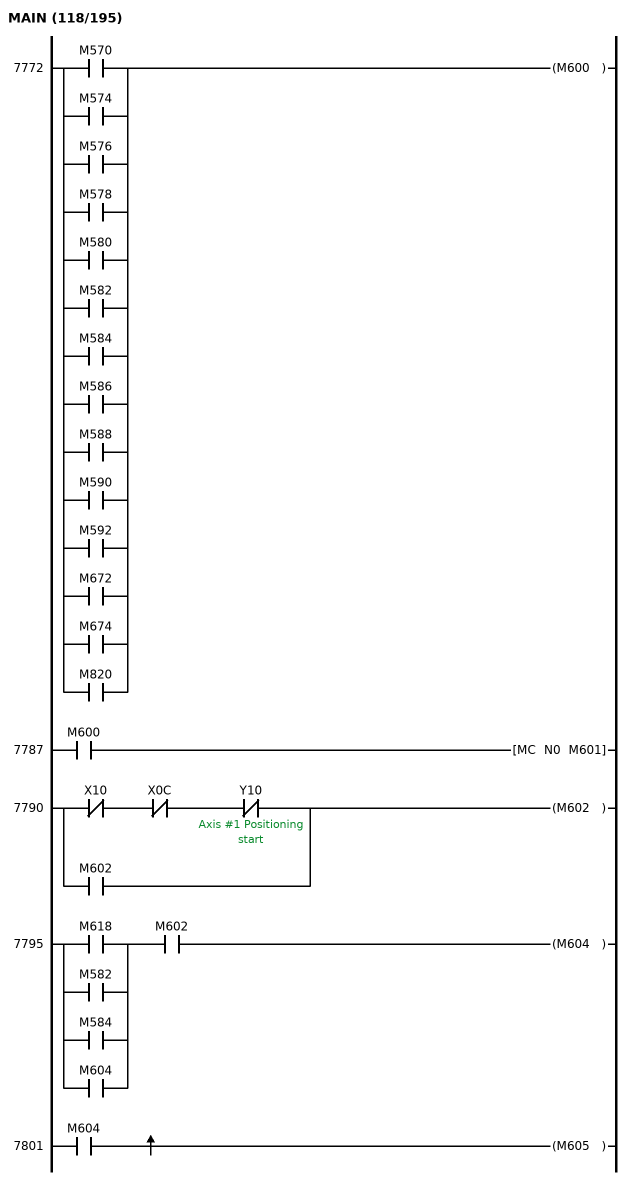
7772  LD      M570
      OR      M574
      OR      M576
      OR      M578
      OR      M580
      OR      M582
      OR      M584
      OR      M586
      OR      M588
      OR      M590
      OR      M592
      OR      M672
      OR      M674
      OR      M820
      OUT     M600
7787  LD      M600
      MC      N0 M601
7790  LDI     X10
      ANI     X0C
      ANI     Y10  ; Axis #1 Positioning start
      OR      M602
      OUT     M602
7795  LD      M618
      OR      M582
      OR      M584
      OR      M604
      AND     M602
      OUT     M604
7801  LD      M604
      MEP
      OUT     M605
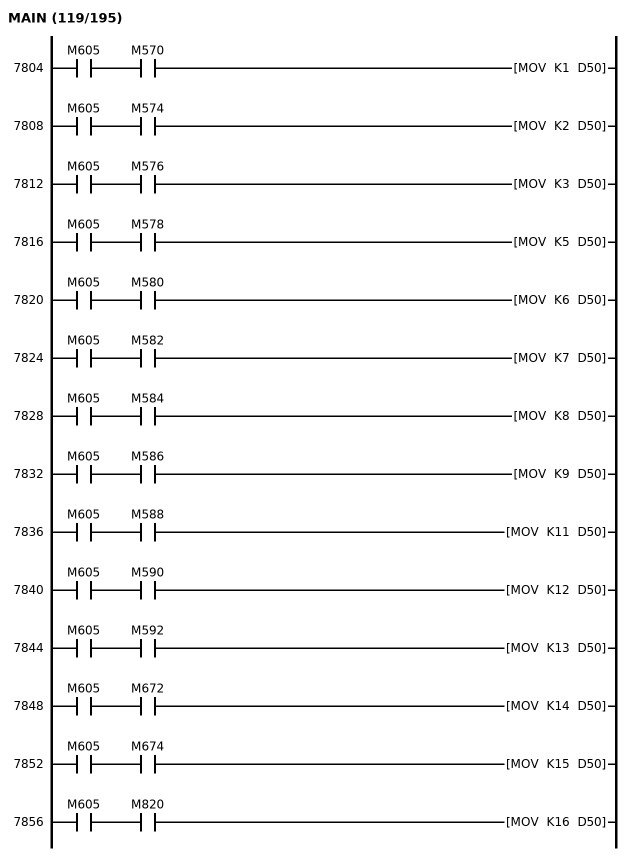
7804  LD      M605
      AND     M570
      MOV     K1 D50
7808  LD      M605
      AND     M574
      MOV     K2 D50
7812  LD      M605
      AND     M576
      MOV     K3 D50
7816  LD      M605
      AND     M578
      MOV     K5 D50
7820  LD      M605
      AND     M580
      MOV     K6 D50
7824  LD      M605
      AND     M582
      MOV     K7 D50
7828  LD      M605
      AND     M584
      MOV     K8 D50
7832  LD      M605
      AND     M586
      MOV     K9 D50
7836  LD      M605
      AND     M588
      MOV     K11 D50
7840  LD      M605
      AND     M590
      MOV     K12 D50
7844  LD      M605
      AND     M592
      MOV     K13 D50
7848  LD      M605
      AND     M672
      MOV     K14 D50
7852  LD      M605
      AND     M674
      MOV     K15 D50
7856  LD      M605
      AND     M820
      MOV     K16 D50
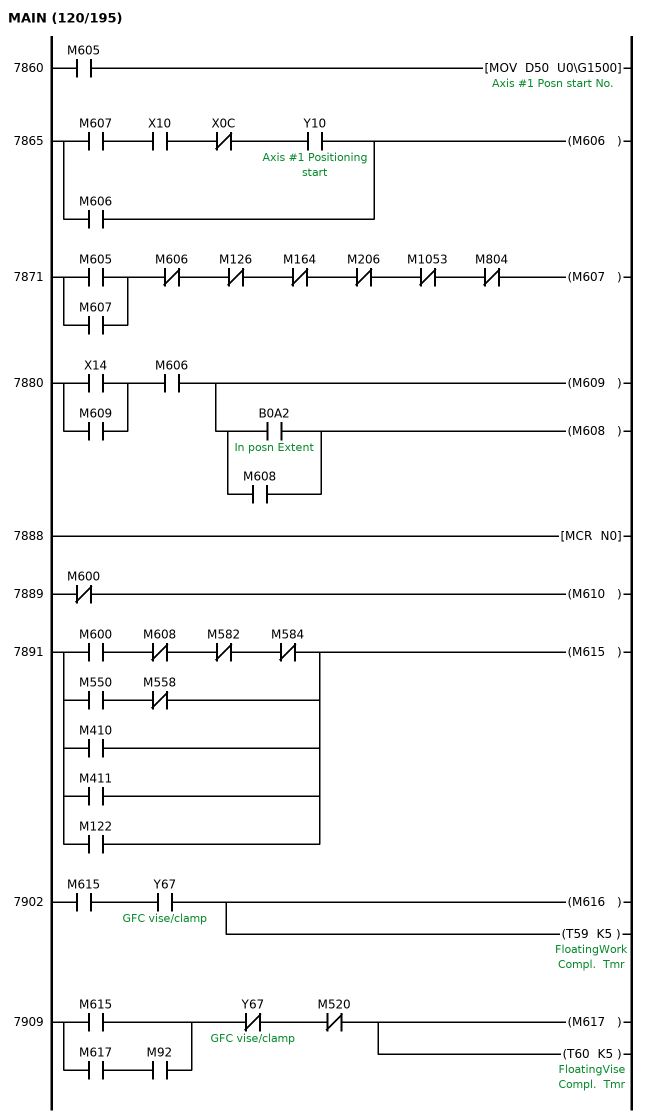
7860  LD      M605
      MOV     D50 U0\G1500  ; Axis #1 Posn start No.
7865  LD      M607
      AND     X10
      ANI     X0C
      AND     Y10  ; Axis #1 Positioning start
      OR      M606
      OUT     M606
7871  LD      M605
      OR      M607
      ANI     M606
      ANI     M126
      ANI     M164
      ANI     M206
      ANI     M1053
      ANI     M804
      OUT     M607
7880  LD      X14
      OR      M609
      AND     M606
      OUT     M609
      LD      B0A2  ; In posn Extent
      OR      M608
      ANB
      OUT     M608
7888  MCR     N0
7889  LDI     M600
      OUT     M610
7891  LD      M600
      ANI     M608
      ANI     M582
      ANI     M584
      LD      M550
      ANI     M558
      ORB
      OR      M410
      OR      M411
      OR      M122
      OUT     M615
7902  LD      M615
      AND     Y67  ; GFC vise/clamp
      OUT     M616
      OUT     T59 K5  ; FloatingWork    Compl.  Tmr
7909  LD      M615
      LD      M617
      AND     M92
      ORB
      ANI     Y67  ; GFC vise/clamp
      ANI     M520
      OUT     M617
      OUT     T60 K5  ; FloatingVise    Compl.  Tmr
